{attribute 'GeneratedUsingTerminal: KL6224-0001'}
{attribute addProperty BoxType "KL6224-0001"}
{attribute addProperty Id "Channel_1AT %Q*Channel_085338040"}
{attribute addProperty CRC "4229837715"}
{attribute addProperty Size "0"}
TYPE KL_FC1E3393 :
STRUCT
	{attribute addProperty Name "Channel_1"}
	Channel_1 : Channel_08533804;
END_STRUCT
END_TYPE

(* stored: Version 1.2.0.0, ProductVersion 3.1.4024.9
   DUT KL_FC1E3393: Id {f3c9edfe-220c-44b6-a09b-12fbde5cd9ae} *)
